TYPE EL3443_Phase_Status :
STRUCT
END_STRUCT
END_TYPE

(* stored: Version 1.1.0.1, ProductVersion 3.1.4024.12
   DUT EL3443_Phase_Status: Id {f8cfb79b-0b82-4ad5-83ef-3a002eff3d81} *)
